{attribute 'GeneratedUsingTerminal: EK1100-0000-0018'}
{attribute addProperty BoxType "EK1100-0000-0018"}
{attribute addProperty Id "Beckhoff_EL29xxEK1122Beckhoff_EL29xxEK1122_F1BDF7ED2A_0001_EL2911_0000_0016EL2911_D6E8124230A_0002_EL2912_0000_0016EL2912_094A1A0A28"}
{attribute addProperty CRC "2202357630"}
{attribute addProperty Size "60"}
TYPE Beckhoff_EL29xx_83454F7E EXTENDS EK1100_1FC0878B :
STRUCT
	{attribute addProperty Name "Beckhoff_EL29xxEK1122"}
	{attribute addProperty PreviousPort "Beckhoff EL29xx : B"}
	Beckhoff_EL29xxEK1122 : Beckhoff_EL29xxEK1122_F1BDF7ED;
	{attribute addProperty Name "A_0001_EL2911_0000_0016"}
	{attribute addProperty PreviousPort "Beckhoff EL29xxEK1122 : C"}
	A_0001_EL2911_0000_0016 : EL2911_D6E81242;
	{attribute addProperty Name "A_0002_EL2912_0000_0016"}
	{attribute addProperty PreviousPort "A_0001(EL2911-0000-0016) : B"}
	A_0002_EL2912_0000_0016 : EL2912_094A1A0A;
END_STRUCT
END_TYPE

(* stored: Version 1.2.0.0, ProductVersion 3.1.4024.9
   DUT Beckhoff_EL29xx_83454F7E: Id {6384653b-54d6-4c7b-a11c-a2226035b935} *)
